// TIA Portal project "instalacja_cieplna_338a_V15_V16" (V16)

(* hardware
DEVICE "GSD device_1"  GSD.Device.PN
   slot 0: "Rack"  Rail  V1.0
   slot 0: "AL1102_2"  AL1102
   slot 1: "8 Ports_1"  AL1102
DEVICE "GSD device_2"  GSD.Device.PN
   slot 0: "Rack"  Rail  V1.0
   slot 0: "AL1102_3"  AL1102
   slot 1: "8 Ports_1"  AL1102
DEVICE "GSD device_3"  GSD.Device.PN
   slot 0: "Rack"  Rail  V1.0
   slot 0: "AL1102_4"  AL1102
   slot 1: "8 Ports_1"  AL1102
   slot 6: "IO-Link In  8 Byte + PQI"  IO-Link In  8 Byte + PQI
   slot 8: "IO-Link In  4 Byte + PQI_1"  IO-Link In  4 Byte + PQI
DEVICE "S71500/ET200MP station_2"  S7-1500 station
   slot 0: "Rail_0"  Rack  6ES7 590-1***0-0AA0
   slot 1: "IO device_1"  IM 155-5 PN HF  6ES7 155-5AA00-0AC0  V3.0
   slot 2: "DQ 32x24VDC/0.5A ST_1"  DQ 32x24VDC/0.5A ST  6ES7 522-1BL00-0AB0  V2.0
   slot 3: "AI 8xU/I/RTD/TC ST_1"  AI 8xU/I/RTD/TC ST  6ES7 531-7KF00-0AB0  V2.0
   slot 4: "AQ 4xU/I ST_1"  AQ 4xU/I ST  6ES7 532-5HD00-0AB0  V2.0
DEVICE "S7-1200 station_1"  S7-1200 Station
   slot 0: "Rack_0"  S7-1200 Rack  Rack  V1.0
   slot 1: "PLC_1"  CPU 1212C DC/DC/DC  6ES7 212-1AE40-0XB0  V4.4
*)

// ===== PLC "PLC_1"  CPU 1212C DC/DC/DC =====

VAR_GLOBAL   // PLC tag table "Default tag table"
   "Heater_PWR_Out" AT %Q0.3 : Bool;
   "Heater_Tout_In" AT %IW127 : Int;   // Temperatura wyjsciowa piec
   "HeatEx_1_Tin_1_In" AT %IW35 : Int;   // Tin wym gora ciepła
   "HeatEx_1_Tout_1_In" AT %IW83 : Int;   // Tout wym gora ciepła
   "Heater_Flow_In" AT %IW112 : Int;   // Przepływ na wejsciu do ogrzewacza
   "HeatEx_1_Flow_In" AT %IW40 : Int;   // przepływ F2
   "Heater_Tin_In" AT %IW103 : Int;   // Temperatura wejściowa piec
   "Heater_Valve_Out" AT %QW8 : Int;   // Wyjście na zawór piec
   "HeatEx_1_Valve_Out" AT %QW4 : Int;   // Wyjscie na zawor wymiennika ciepla góra
   "HeatEx_1_Tin_2_In" AT %IW78 : Int;   // Tin wym gora zimna
   "HeatEx_1_Tout_2_In" AT %IW30 : Int;   // Tout wym gora zimna
   "HeatEx_2_Tin_2_In" AT %IW73 : Int;   // Tin wym dol zimna
   "HeatEx_2_Tin_1_In" AT %IW68 : Int;   // Tin wym dol ciepła
   "HeatEx_2_Tout_2_In" AT %IW122 : Int;   // Tout wym dol zimna
   "HeatEx_2_ValveOut" AT %QW6 : Int;   // wyjście na zawór wymiennika ciepła dół
   "HeatEx_2_Flow_In" AT %IW49 : Int;   // przepływ F3
   "Preassure_In" AT %IW132 : Int;   // Cisnienie wejsciowe na piec
   "off" AT %M0.0 : Bool;
   "start" AT %M0.1 : Bool;
   "reset" AT %M0.2 : Bool;
   "dist" AT %MD2 : Real;
   "dist_SP" AT %MD6 : Real;
   "test" AT %MD10 : Real;
   "step_dist" AT %MD14 : Real;
   "HeatEx_SP" AT %MD18 : Real;
   "HeatEx_2_Tout1_In" AT %IW98 : Int;   // Tout wym dol ciepła
   "Always_OFF" AT %M0.3 : Bool;
   "Preassure_HeatEx_In" AT %IW11 : Int;
   "Preassure_HeatEx_Out" AT %IW17 : Int;
   "Tag_1" AT %QW1 : Int;
   "Tag_2" AT %QW0 : Int;
END_VAR

VAR_GLOBAL CONSTANT   // PLC tag table "Default tag table"
   "None(1)" : Pip := 65535;
   "Automatic update(1)" : Pip := 0;
   "PIP 1(1)" : Pip := 1;
   "PIP 2(1)" : Pip := 2;
   "PIP 3(1)" : Pip := 3;
   "PIP 4(1)" : Pip := 4;
   "PIP 5" : Pip := 5;
   "PIP 6" : Pip := 6;
   "PIP 7" : Pip := 7;
   "PIP 8" : Pip := 8;
   "PIP 9" : Pip := 9;
   "PIP 10" : Pip := 10;
   "PIP 11" : Pip := 11;
   "PIP 12" : Pip := 12;
   "PIP 13" : Pip := 13;
   "PIP 14" : Pip := 14;
   "PIP 15" : Pip := 15;
   "PIP 16" : Pip := 16;
   "PIP 17" : Pip := 17;
   "PIP 18" : Pip := 18;
   "PIP 19" : Pip := 19;
   "PIP 20" : Pip := 20;
   "PIP 21" : Pip := 21;
   "PIP 22" : Pip := 22;
   "PIP 23" : Pip := 23;
   "PIP 24" : Pip := 24;
   "PIP 25" : Pip := 25;
   "PIP 26" : Pip := 26;
   "PIP 27" : Pip := 27;
   "PIP 28" : Pip := 28;
   "PIP 29" : Pip := 29;
   "PIP 30" : Pip := 30;
   "PIP 31" : Pip := 31;
   "PIP OB Servo(1)" : Pip := 32768;
   "Local~Common(1)" : Hw_SubModule := 50;
   "Local(1)" : Hw_SubModule := 49;
   "OB_Main(1)" : OB_PCYCLE := 1;
   "Local~Display" : Hw_SubModule := 54;
   "Local~MC(1)" : Hw_SubModule := 51;
   "Local~Exec(1)" : Hw_SubModule := 52;
   "Local~PROFINET_interface_1(1)" : Hw_Interface := 64;
   "Local~PROFINET_interface_1~Port_1(1)" : Hw_Interface := 65;
   "Local~PROFINET_interface_1~Port_2" : Hw_Interface := 66;
   "Local~PROFINET_IO-System" : Hw_IoSystem := 257;
   "AL1102_4~Proxy" : Hw_SubModule := 310;
   "AL1102_4~IODevice" : Hw_Device := 308;
   "AL1102_4~X1" : Hw_Interface := 311;
   "AL1102_4~X1~Port_1" : Hw_Interface := 312;
   "AL1102_4~X1~Port_2" : Hw_Interface := 283;
   "AL1102_4~Head" : Hw_SubModule := 284;
   "AL1102_4~8_Ports_1~IO-Link_Master" : Hw_SubModule := 286;
   "AL1102_4~8_Ports_1" : Hw_SubModule := 303;
   "AL1102_4~8_Ports_1~IO-Link_In__4_Byte_+_PQI" : Hw_SubModule := 304;
   "AL1102_4~8_Ports_1~IO-Link_In__8_Byte_+_PQI" : Hw_SubModule := 305;
   "AL1102_4~8_Ports_1~IO-Link_In__4_Byte_+_PQI_2" : Hw_SubModule := 307;
   "AL1102_3~Proxy" : Hw_SubModule := 280;
   "AL1102_3~IODevice" : Hw_Device := 278;
   "AL1102_3~X1" : Hw_Interface := 281;
   "AL1102_3~X1~Port_1" : Hw_Interface := 282;
   "AL1102_3~X1~Port_2" : Hw_Interface := 276;
   "AL1102_3~Head" : Hw_SubModule := 277;
   "AL1102_3~8_Ports_1~IO-Link_Master" : Hw_SubModule := 287;
   "AL1102_3~8_Ports_1" : Hw_SubModule := 292;
   "AL1102_3~8_Ports_1~IO-Link_In__8_Byte_+_PQI" : Hw_SubModule := 293;
   "AL1102_3~8_Ports_1~IO-Link_In__8_Byte_+_PQI_1" : Hw_SubModule := 294;
   "AL1102_3~8_Ports_1~IO-Link_In__4_Byte_+_PQI" : Hw_SubModule := 295;
   "AL1102_3~8_Ports_1~IO-Link_In__4_Byte_+_PQI_1" : Hw_SubModule := 296;
   "AL1102_3~8_Ports_1~IO-Link_In__4_Byte_+_PQI_2" : Hw_SubModule := 297;
   "AL1102_3~8_Ports_1~IO-Link_In__4_Byte_+_PQI_3" : Hw_SubModule := 298;
   "AL1102_2~Proxy" : Hw_SubModule := 273;
   "AL1102_2~IODevice" : Hw_Device := 271;
   "AL1102_2~PROFINET_interface_1" : Hw_Interface := 274;
   "AL1102_2~PROFINET_interface_1~Port_1" : Hw_Interface := 268;
   "AL1102_2~PROFINET_interface_1~Port_2" : Hw_Interface := 269;
   "AL1102_2~Head" : Hw_SubModule := 270;
   "AL1102_2~8_Ports_1~IO-Link_Master" : Hw_SubModule := 275;
   "AL1102_2~8_Ports_1~IO-Link_In__4_Byte_+_PQI" : Hw_SubModule := 288;
   "AL1102_2~8_Ports_1" : Hw_SubModule := 285;
   "AL1102_2~8_Ports_1~IO-Link_In__4_Byte_+_PQI_1" : Hw_SubModule := 289;
   "AL1102_2~8_Ports_1~IO-Link_In__4_Byte_+_PQI_2" : Hw_SubModule := 290;
   "AL1102_2~8_Ports_1~IO-Link_In__4_Byte_+_PQI_3" : Hw_SubModule := 291;
   "AL1102_2~8_Ports_1~IO-Link_In__4_Byte_+_PQI_4" : Hw_SubModule := 299;
   "AL1102_2~8_Ports_1~IO-Link_In__4_Byte_+_PQI_5" : Hw_SubModule := 300;
   "AL1102_2~8_Ports_1~IO-Link_In__4_Byte_+_PQI_7" : Hw_SubModule := 302;
   "IO_device_1~Proxy" : Hw_SubModule := 315;
   "IO_device_1~IODevice" : Hw_Device := 313;
   "IO_device_1~PROFINET_interface" : Hw_Interface := 316;
   "IO_device_1~PROFINET_interface~Port_1" : Hw_Interface := 317;
   "IO_device_1~PROFINET_interface~Port_2" : Hw_Interface := 318;
   "IO_device_1~Head" : Hw_SubModule := 319;
   "IO_device_1~DQ_32x24VDC_0_5A_ST_1" : Hw_SubModule := 320;
   "IO_device_1~AI_8xU_I_RTD_TC_ST_1" : Hw_SubModule := 321;
   "IO_device_1~AQ_4xU_I_ST_1" : Hw_SubModule := 322;
   "OB_Startup(1)" : OB_STARTUP := 100;
   "OB_Flow controllers(1)" : OB_Cyclic := 30;
END_VAR

DATA_BLOCK "Signals_DB"   // DB3
{ S7_Optimized_Access := 'TRUE' }
VERSION : 0.1
   VAR
      Heater_Tout_PIDOut : Real;
      Heater_Tout_SP : Real;
      PWM_period : Int;
      PIorPID : Bool;   // 0 - PI, 1 - PID
      Heater_PWR : Real;
      Heater_Alarm : Bool;
      Heater_ResetAlarm : Bool;
      Heater_Tin : Real;
   END_VAR
   VAR RETAIN
      Heater_Tout : Real;
   END_VAR
   VAR
      HeatEx_1_Tin_1 : Real;
      HeatEx_1_Tin_2 : Real;
      HeatEx_1_Tout_1 : Real;
      HeatEx_1_Tout_2 : Real;
      HeatEx_2_Tin_1 : Real;
      HeatEx_2_Tin_2 : Real;
      HeatEx_2_Tout_1 : Real;
      HeatEx_2_Tout_2 : Real;
      Heater_Flow : Real;
      HeatEx_1_Flow : Real;
      HeatEx_2_Flow : Real;
      Heater_Flow_SP : Real;
      Heater_Valve : Real;
      Preassure : Real;
      Preassure_HeatEx_In : Real;
      Preassure_HeatEx_Out : Real;
      HeatEx_1_Flow_SP : Real;
      HeatEx_1_Valve : Real;
      HeatEx_2_FlowSP : Real;
      HeatEx_2_Valve : Real;
      AutoOrManual : Bool;   // Manual = true, Auto = false
      Tout_setpoint : Real;
      PIDMode : Int := 3;
   END_VAR
BEGIN
END_DATA_BLOCK

DATA_BLOCK "PWM_DB"   // DB6
{ S7_Optimized_Access := 'TRUE' }
VERSION : 0.1
// stored: InstanceOfName PWM
"PWM"
BEGIN
END_DATA_BLOCK

DATA_BLOCK "Signals_to_S7protocol"   // DB8
{ S7_Optimized_Access := 'FALSE' }
VERSION : 0.1
   VAR
      OUT : Struct   // PLC out going to Raspbery
         Heater_Tout_setpoint : Real;   // Setpoint output temperature [°C]
         Heater_Flow_actual : Real;   // Actual flow [l/min]
         Heater_Flow_setpoint : Real;   // Flow setpoint[l/min]
         Auto_Or_Manual : Bool;   // Auto - true MAnual - false
         Heater_Tout_actual : Real;   // Actual output temperature [°C]
         Heater_Power_setpoint : Real;   // Percentage heater power rate 0-100
         Counter_OUT : Int;   // Output counter to Raspberry PI
      END_STRUCT;
      IN : Struct   // PLC in from Raspberry
         Flow_setpoint : Real;   // Flow setpoint [l/min]
         Counter_IN : Int;   // Input ciunter from Raspberry PI
      END_STRUCT;
      IN_OUT : Struct
         LiveBit : Bool;   // Communication LiveBit setting in each cycle of OB32
      END_STRUCT;
      INTERNAL : Struct
         Communication_Error : Bool;   // Communication error alarm
         Count_Up_Each_Cycle : Bool;
      END_STRUCT;
   END_VAR
BEGIN
END_DATA_BLOCK

// folder: System blocks/Program resources

DATA_BLOCK "IEC_Timer_0_DB"   // DB1
{ S7_Optimized_Access := 'TRUE' }
AUTHOR : Simatic
FAMILY : IEC
NAME : IEC_TMR
VERSION : 1.0
// stored: InstanceOfName IEC_TIMER
"IEC_TIMER"
BEGIN
END_DATA_BLOCK

DATA_BLOCK "IEC_Timer_0_DB_1"   // DB2
{ S7_Optimized_Access := 'TRUE' }
AUTHOR : Simatic
FAMILY : IEC
NAME : IEC_TMR
VERSION : 1.0
// stored: InstanceOfName IEC_TIMER
"IEC_TIMER"
BEGIN
END_DATA_BLOCK

DATA_BLOCK "LiveBit_timer"   // DB9
{ S7_Optimized_Access := 'TRUE' }
AUTHOR : Simatic
FAMILY : IEC
NAME : IEC_TMR
VERSION : 1.0
// stored: InstanceOfName IEC_TIMER
"IEC_TIMER"
BEGIN
END_DATA_BLOCK

DATA_BLOCK "Communication_Couter"   // DB10
{ S7_Optimized_Access := 'TRUE' }
AUTHOR : Simatic
FAMILY : IEC
NAME : CNTR
VERSION : 1.0
// stored: InstanceOfName IEC_COUNTER
"IEC_COUNTER"
BEGIN
END_DATA_BLOCK

// folder: (top level)

FUNCTION_BLOCK "PWM"   // FB2, LAD
{ S7_Optimized_Access := 'TRUE' }
VERSION : 0.1
   VAR_INPUT
      width : Int;
      cycle : Int;
   END_VAR
   VAR_IN_OUT
      output : Bool;
   END_VAR
   VAR_TEMP
      T1 : Int;
      T2 : Int;
      czas1 : Time;
      czas2 : Time;
   END_VAR
BEGIN

REGION Network 1: Obliczanie T1 i T2 na podstawie czasu cyklu i szerokości impulsu
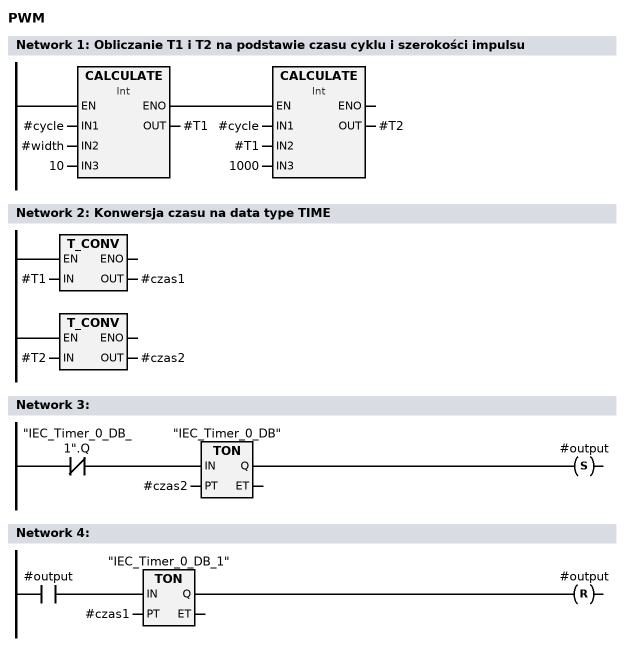
   RUNG wire#powerrail
      { S7_Templates := "SrcType := Int"; S7_GenerateENO := "TRUE"; S7_Expression := "IN1*IN2*IN3" } Calculate(in1 := #cycle, in2 := #width, in3 := 10, out => #T1)
      { S7_Templates := "SrcType := Int"; S7_GenerateENO := "TRUE"; S7_Expression := "IN1*IN3-IN2" } Calculate(in1 := #cycle, in2 := #T1, in3 := 1000, out => #T2)
   END_RUNG
   // the same network as SCL:
   // ENO of a box is taken as its EN; it also drops when the box reports an error
   #T1 := #cycle*#width*10;
   #T2 := #cycle*1000-#T1;
END_REGION

REGION Network 2: Konwersja czasu na data type TIME
   #czas1 := T_CONV(IN := #T1);
   #czas2 := T_CONV(IN := #T2);
END_REGION

REGION Network 3
   "IEC_Timer_0_DB".TON(IN := NOT "IEC_Timer_0_DB_1".Q, PT := #czas2);
   IF "IEC_Timer_0_DB".Q THEN #output := TRUE; END_IF;
END_REGION

REGION Network 4
   "IEC_Timer_0_DB_1".TON(IN := #output, PT := #czas1);
   IF "IEC_Timer_0_DB_1".Q THEN #output := FALSE; END_IF;
END_REGION
END_FUNCTION_BLOCK

ORGANIZATION_BLOCK "Main"   // OB1, LAD, ProgramCycle
TITLE = "Main Program Sweep (Cycle)"
{ S7_Optimized_Access := 'TRUE' }
VERSION : 0.1
   VAR_INPUT
      Initial_Call : Bool;   // Initial call of this OB
      Remanence : Bool;   // =True, if remanent data are available
   END_VAR
   VAR_TEMP
      power_SP_int : Int;
      ret_value : Int;
      scale_press_Heat_Ex_OUT : Real;
      scale_press_PressureIN : Real;
      scale_press_Heat_Ex_IN : Real;
      unscale_Heater_Valve : Real;
      unscale_HeatEX_2_ValveOut : Real;
      unscale_HeatEX_1_ValveOut : Real;
      tmp_PID_Tout_Rate : Real;
   END_VAR
BEGIN

REGION Network 1: Sterowanie mocą pieca
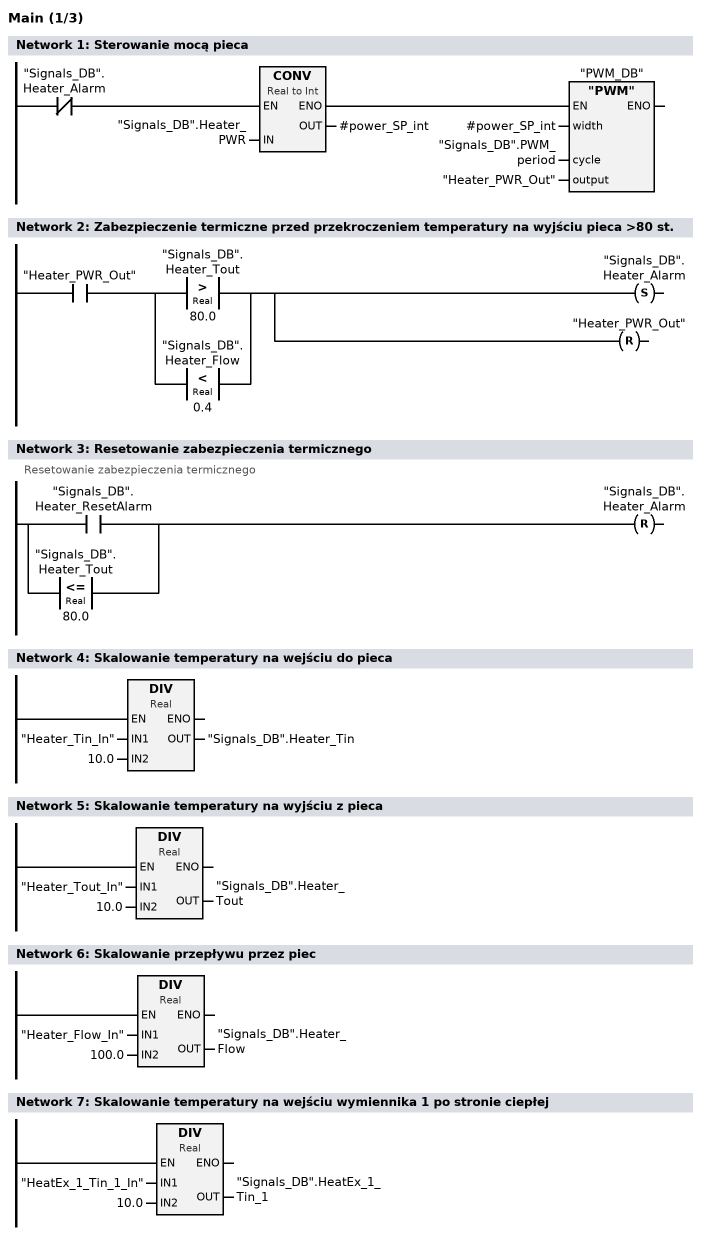
   RUNG wire#powerrail
      I_Contact( "Signals_DB".Heater_Alarm )
      { S7_Templates := "[SrcType := Real, DestType := Int]"; S7_GenerateENO := "TRUE" } Convert(in := "Signals_DB".Heater_PWR, out => #power_SP_int)
      "PWM_DB"(width := #power_SP_int, cycle := "Signals_DB".PWM_period, output := "Heater_PWR_Out")
   END_RUNG
   // the same network as SCL:
   // ENO of a box is taken as its EN; it also drops when the box reports an error
   IF NOT "Signals_DB".Heater_Alarm THEN
       #power_SP_int := REAL_TO_INT("Signals_DB".Heater_PWR);
       "PWM_DB"(width := #power_SP_int, cycle := "Signals_DB".PWM_period, output := "Heater_PWR_Out");   // "PWM"
   END_IF;
END_REGION

REGION Network 2: Zabezpieczenie termiczne przed przekroczeniem temperatury na wyjściu pieca >80 st.
   RUNG wire#powerrail
      Contact( "Heater_PWR_Out" )
      wire#w1
      { S7_Templates := "SrcType := Real" } GT_Contact(in1 := "Signals_DB".Heater_Tout, in2 := 80.0)
      wire#w2
      S_Coil( "Signals_DB".Heater_Alarm )
   END_RUNG
   RUNG wire#w1
      { S7_Templates := "SrcType := Real" } LT_Contact(in1 := "Signals_DB".Heater_Flow, in2 := 0.4)
   END_RUNG wire#w2
   RUNG wire#w2
      R_Coil( "Heater_PWR_Out" )
   END_RUNG
   // the same network as SCL:
   IF "Heater_PWR_Out" AND (("Signals_DB".Heater_Tout > 80.0) OR ("Signals_DB".Heater_Flow < 0.4)) THEN
       "Signals_DB".Heater_Alarm := TRUE;
       "Heater_PWR_Out" := FALSE;
   END_IF;
END_REGION

REGION Network 3: Resetowanie zabezpieczenia termicznego
   // Resetowanie zabezpieczenia termicznego
   RUNG wire#powerrail
      Contact( "Signals_DB".Heater_ResetAlarm )
      wire#w1
      R_Coil( "Signals_DB".Heater_Alarm )
   END_RUNG
   RUNG wire#powerrail
      { S7_Templates := "SrcType := Real" } LE_Contact(in1 := "Signals_DB".Heater_Tout, in2 := 80.0)
   END_RUNG wire#w1
   // the same network as SCL:
   IF "Signals_DB".Heater_ResetAlarm OR ("Signals_DB".Heater_Tout <= 80.0) THEN
       "Signals_DB".Heater_Alarm := FALSE;
   END_IF;
END_REGION

REGION Network 4: Skalowanie temperatury na wejściu do pieca
   RUNG wire#powerrail
      { S7_Templates := "SrcType := Real"; S7_GenerateENO := "TRUE" } Div(in1 := "Heater_Tin_In", in2 := 10.0, out => "Signals_DB".Heater_Tin)
   END_RUNG
   // the same network as SCL:
   "Signals_DB".Heater_Tin := "Heater_Tin_In" / 10.0;
END_REGION

REGION Network 5: Skalowanie temperatury na wyjściu z pieca
   RUNG wire#powerrail
      { S7_Templates := "SrcType := Real"; S7_GenerateENO := "TRUE" } Div(in1 := "Heater_Tout_In", in2 := 10.0, out => "Signals_DB".Heater_Tout)
   END_RUNG
   // the same network as SCL:
   "Signals_DB".Heater_Tout := "Heater_Tout_In" / 10.0;
END_REGION

REGION Network 6: Skalowanie przepływu przez piec
   RUNG wire#powerrail
      { S7_Templates := "SrcType := Real"; S7_GenerateENO := "TRUE" } Div(in1 := "Heater_Flow_In", in2 := 100.0, out => "Signals_DB".Heater_Flow)
   END_RUNG
   // the same network as SCL:
   "Signals_DB".Heater_Flow := "Heater_Flow_In" / 100.0;
END_REGION

REGION Network 7: Skalowanie temperatury na wejściu wymiennika 1 po stronie ciepłej
   RUNG wire#powerrail
      { S7_Templates := "SrcType := Real"; S7_GenerateENO := "TRUE" } Div(in1 := "HeatEx_1_Tin_1_In", in2 := 10.0, out => "Signals_DB".HeatEx_1_Tin_1)
   END_RUNG
   // the same network as SCL:
   "Signals_DB".HeatEx_1_Tin_1 := "HeatEx_1_Tin_1_In" / 10.0;
END_REGION

REGION Network 8: Skalowanie temperatury na wyjściu z wymiennika 1 po stronie ciepłej
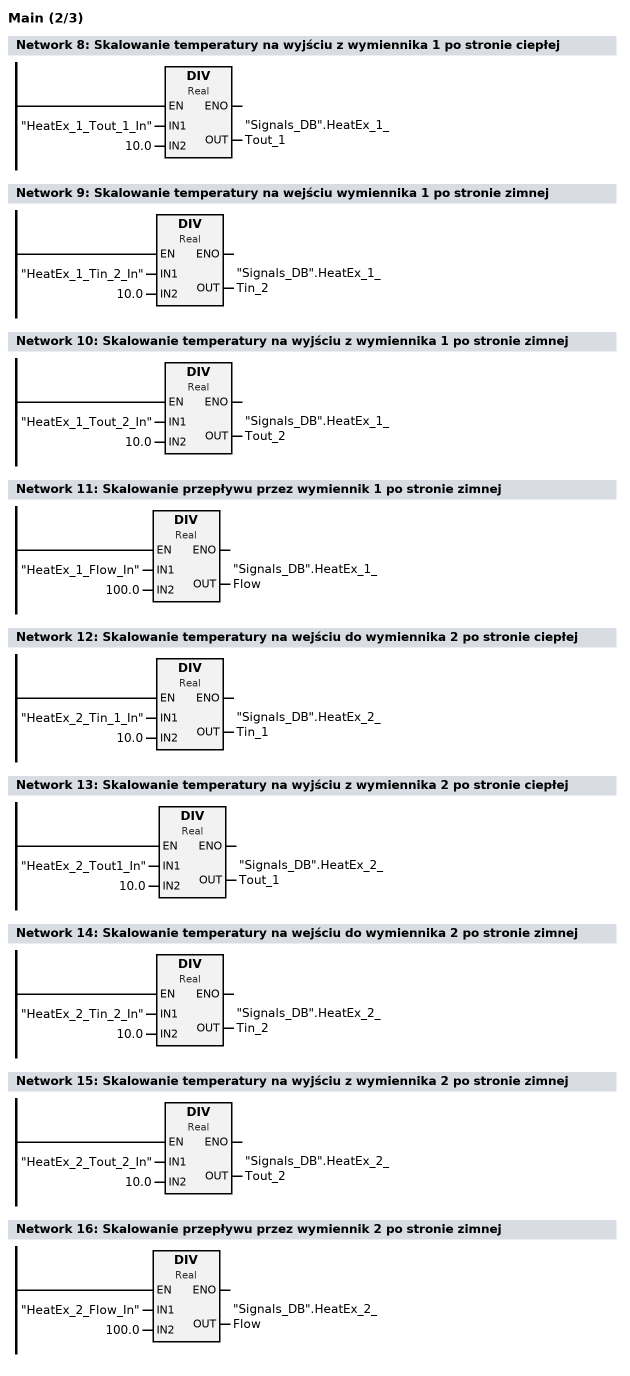
   RUNG wire#powerrail
      { S7_Templates := "SrcType := Real"; S7_GenerateENO := "TRUE" } Div(in1 := "HeatEx_1_Tout_1_In", in2 := 10.0, out => "Signals_DB".HeatEx_1_Tout_1)
   END_RUNG
   // the same network as SCL:
   "Signals_DB".HeatEx_1_Tout_1 := "HeatEx_1_Tout_1_In" / 10.0;
END_REGION

REGION Network 9: Skalowanie temperatury na wejściu wymiennika 1 po stronie zimnej
   RUNG wire#powerrail
      { S7_Templates := "SrcType := Real"; S7_GenerateENO := "TRUE" } Div(in1 := "HeatEx_1_Tin_2_In", in2 := 10.0, out => "Signals_DB".HeatEx_1_Tin_2)
   END_RUNG
   // the same network as SCL:
   "Signals_DB".HeatEx_1_Tin_2 := "HeatEx_1_Tin_2_In" / 10.0;
END_REGION

REGION Network 10: Skalowanie temperatury na wyjściu z wymiennika 1 po stronie zimnej
   RUNG wire#powerrail
      { S7_Templates := "SrcType := Real"; S7_GenerateENO := "TRUE" } Div(in1 := "HeatEx_1_Tout_2_In", in2 := 10.0, out => "Signals_DB".HeatEx_1_Tout_2)
   END_RUNG
   // the same network as SCL:
   "Signals_DB".HeatEx_1_Tout_2 := "HeatEx_1_Tout_2_In" / 10.0;
END_REGION

REGION Network 11: Skalowanie przepływu przez wymiennik 1 po stronie zimnej
   RUNG wire#powerrail
      { S7_Templates := "SrcType := Real"; S7_GenerateENO := "TRUE" } Div(in1 := "HeatEx_1_Flow_In", in2 := 100.0, out => "Signals_DB".HeatEx_1_Flow)
   END_RUNG
   // the same network as SCL:
   "Signals_DB".HeatEx_1_Flow := "HeatEx_1_Flow_In" / 100.0;
END_REGION

REGION Network 12: Skalowanie temperatury na wejściu do wymiennika 2 po stronie ciepłej
   RUNG wire#powerrail
      { S7_Templates := "SrcType := Real"; S7_GenerateENO := "TRUE" } Div(in1 := "HeatEx_2_Tin_1_In", in2 := 10.0, out => "Signals_DB".HeatEx_2_Tin_1)
   END_RUNG
   // the same network as SCL:
   "Signals_DB".HeatEx_2_Tin_1 := "HeatEx_2_Tin_1_In" / 10.0;
END_REGION

REGION Network 13: Skalowanie temperatury na wyjściu z wymiennika 2 po stronie ciepłej
   RUNG wire#powerrail
      { S7_Templates := "SrcType := Real"; S7_GenerateENO := "TRUE" } Div(in1 := "HeatEx_2_Tout1_In", in2 := 10.0, out => "Signals_DB".HeatEx_2_Tout_1)
   END_RUNG
   // the same network as SCL:
   "Signals_DB".HeatEx_2_Tout_1 := "HeatEx_2_Tout1_In" / 10.0;
END_REGION

REGION Network 14: Skalowanie temperatury na wejściu do wymiennika 2 po stronie zimnej
   RUNG wire#powerrail
      { S7_Templates := "SrcType := Real"; S7_GenerateENO := "TRUE" } Div(in1 := "HeatEx_2_Tin_2_In", in2 := 10.0, out => "Signals_DB".HeatEx_2_Tin_2)
   END_RUNG
   // the same network as SCL:
   "Signals_DB".HeatEx_2_Tin_2 := "HeatEx_2_Tin_2_In" / 10.0;
END_REGION

REGION Network 15: Skalowanie temperatury na wyjściu z wymiennika 2 po stronie zimnej
   RUNG wire#powerrail
      { S7_Templates := "SrcType := Real"; S7_GenerateENO := "TRUE" } Div(in1 := "HeatEx_2_Tout_2_In", in2 := 10.0, out => "Signals_DB".HeatEx_2_Tout_2)
   END_RUNG
   // the same network as SCL:
   "Signals_DB".HeatEx_2_Tout_2 := "HeatEx_2_Tout_2_In" / 10.0;
END_REGION

REGION Network 16: Skalowanie przepływu przez wymiennik 2 po stronie zimnej
   RUNG wire#powerrail
      { S7_Templates := "SrcType := Real"; S7_GenerateENO := "TRUE" } Div(in1 := "HeatEx_2_Flow_In", in2 := 100.0, out => "Signals_DB".HeatEx_2_Flow)
   END_RUNG
   // the same network as SCL:
   "Signals_DB".HeatEx_2_Flow := "HeatEx_2_Flow_In" / 100.0;
END_REGION

REGION Network 17: Unskalowanie otwarcia zaworu wyjściowego z pieca
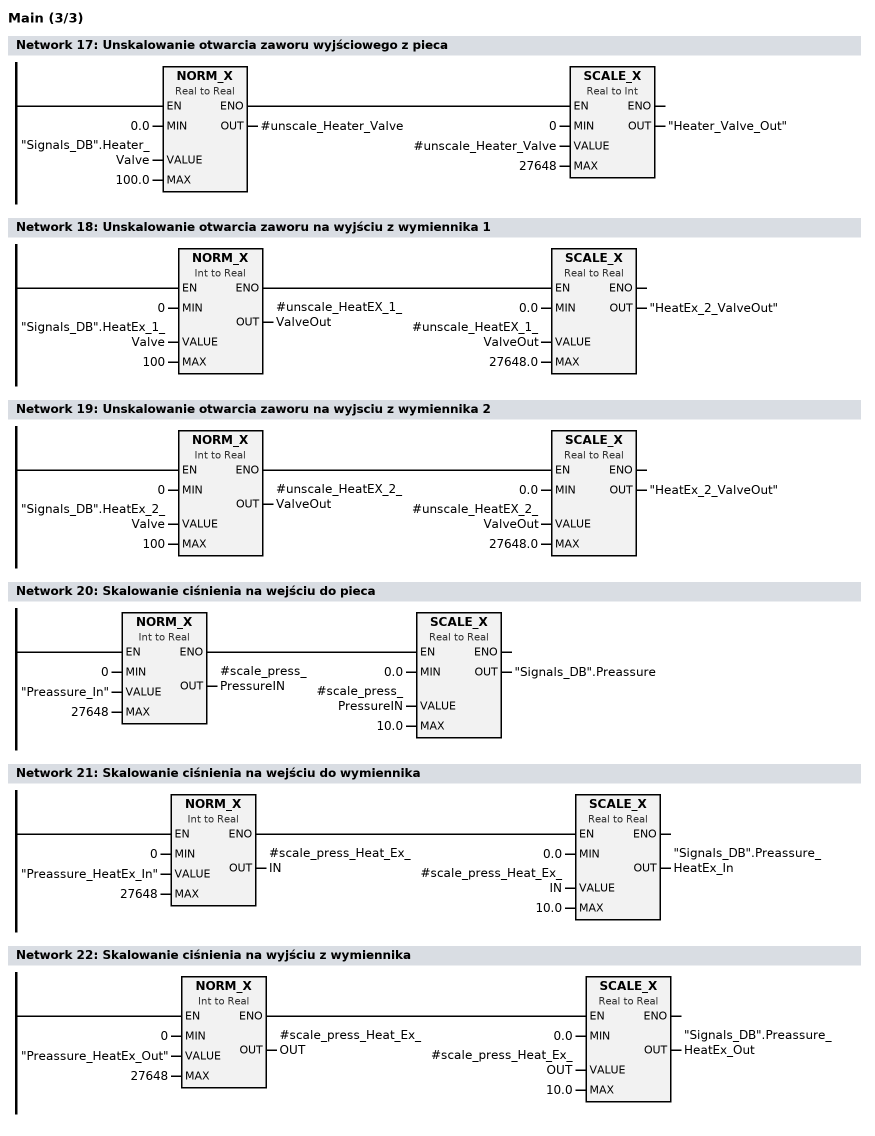
   RUNG wire#powerrail
      { S7_Templates := "[SrcType := Real, DestType := Real]" } Normalize(min := 0.0, value := "Signals_DB".Heater_Valve, max := 100.0, out => #unscale_Heater_Valve)
      { S7_Templates := "[SrcType := Real, DestType := Int]" } Scale(min := 0, value := #unscale_Heater_Valve, max := 27648, out => "Heater_Valve_Out")
   END_RUNG
   // the same network as SCL:
   #unscale_Heater_Valve := NORM_X(MIN := 0.0, VALUE := "Signals_DB".Heater_Valve, MAX := 100.0);
   "Heater_Valve_Out" := SCALE_X(MIN := 0, VALUE := #unscale_Heater_Valve, MAX := 27648);
END_REGION

REGION Network 18: Unskalowanie otwarcia zaworu na wyjściu z wymiennika 1
   RUNG wire#powerrail
      { S7_Templates := "[SrcType := Int, DestType := Real]" } Normalize(min := 0, value := "Signals_DB".HeatEx_1_Valve, max := 100, out => #unscale_HeatEX_1_ValveOut)
      { S7_Templates := "[SrcType := Real, DestType := Real]" } Scale(min := 0.0, value := #unscale_HeatEX_1_ValveOut, max := 27648.0, out => "HeatEx_2_ValveOut")
   END_RUNG
   // the same network as SCL:
   #unscale_HeatEX_1_ValveOut := NORM_X(MIN := 0, VALUE := "Signals_DB".HeatEx_1_Valve, MAX := 100);
   "HeatEx_2_ValveOut" := SCALE_X(MIN := 0.0, VALUE := #unscale_HeatEX_1_ValveOut, MAX := 27648.0);
END_REGION

REGION Network 19: Unskalowanie otwarcia zaworu na wyjsciu z wymiennika 2
   RUNG wire#powerrail
      { S7_Templates := "[SrcType := Int, DestType := Real]" } Normalize(min := 0, value := "Signals_DB".HeatEx_2_Valve, max := 100, out => #unscale_HeatEX_2_ValveOut)
      { S7_Templates := "[SrcType := Real, DestType := Real]" } Scale(min := 0.0, value := #unscale_HeatEX_2_ValveOut, max := 27648.0, out => "HeatEx_2_ValveOut")
   END_RUNG
   // the same network as SCL:
   #unscale_HeatEX_2_ValveOut := NORM_X(MIN := 0, VALUE := "Signals_DB".HeatEx_2_Valve, MAX := 100);
   "HeatEx_2_ValveOut" := SCALE_X(MIN := 0.0, VALUE := #unscale_HeatEX_2_ValveOut, MAX := 27648.0);
END_REGION

REGION Network 20: Skalowanie ciśnienia na wejściu do pieca
   RUNG wire#powerrail
      { S7_Templates := "[SrcType := Int, DestType := Real]" } Normalize(min := 0, value := "Preassure_In", max := 27648, out => #scale_press_PressureIN)
      { S7_Templates := "[SrcType := Real, DestType := Real]" } Scale(min := 0.0, value := #scale_press_PressureIN, max := 10.0, out => "Signals_DB".Preassure)
   END_RUNG
   // the same network as SCL:
   #scale_press_PressureIN := NORM_X(MIN := 0, VALUE := "Preassure_In", MAX := 27648);
   "Signals_DB".Preassure := SCALE_X(MIN := 0.0, VALUE := #scale_press_PressureIN, MAX := 10.0);
END_REGION

REGION Network 21: Skalowanie ciśnienia na wejściu do wymiennika
   RUNG wire#powerrail
      { S7_Templates := "[SrcType := Int, DestType := Real]" } Normalize(min := 0, value := "Preassure_HeatEx_In", max := 27648, out => #scale_press_Heat_Ex_IN)
      { S7_Templates := "[SrcType := Real, DestType := Real]" } Scale(min := 0.0, value := #scale_press_Heat_Ex_IN, max := 10.0, out => "Signals_DB".Preassure_HeatEx_In)
   END_RUNG
   // the same network as SCL:
   #scale_press_Heat_Ex_IN := NORM_X(MIN := 0, VALUE := "Preassure_HeatEx_In", MAX := 27648);
   "Signals_DB".Preassure_HeatEx_In := SCALE_X(MIN := 0.0, VALUE := #scale_press_Heat_Ex_IN, MAX := 10.0);
END_REGION

REGION Network 22: Skalowanie ciśnienia na wyjściu z wymiennika
   RUNG wire#powerrail
      { S7_Templates := "[SrcType := Int, DestType := Real]" } Normalize(min := 0, value := "Preassure_HeatEx_Out", max := 27648, out => #scale_press_Heat_Ex_OUT)
      { S7_Templates := "[SrcType := Real, DestType := Real]" } Scale(min := 0.0, value := #scale_press_Heat_Ex_OUT, max := 10.0, out => "Signals_DB".Preassure_HeatEx_Out)
   END_RUNG
   // the same network as SCL:
   #scale_press_Heat_Ex_OUT := NORM_X(MIN := 0, VALUE := "Preassure_HeatEx_Out", MAX := 27648);
   "Signals_DB".Preassure_HeatEx_Out := SCALE_X(MIN := 0.0, VALUE := #scale_press_Heat_Ex_OUT, MAX := 10.0);
END_REGION
END_ORGANIZATION_BLOCK

ORGANIZATION_BLOCK "Flow controllers"   // OB30, LAD, CyclicInterrupt
{ S7_Optimized_Access := 'TRUE' }
VERSION : 0.1
   VAR_INPUT
      Initial_Call : Bool;   // Initial call of this OB
      Event_Count : Int;   // Events discarded
   END_VAR
   VAR_TEMP
      PIorPID : Bool;
   END_VAR
BEGIN

REGION Network 1: PID do sterowania nagrzewaniem cieczy
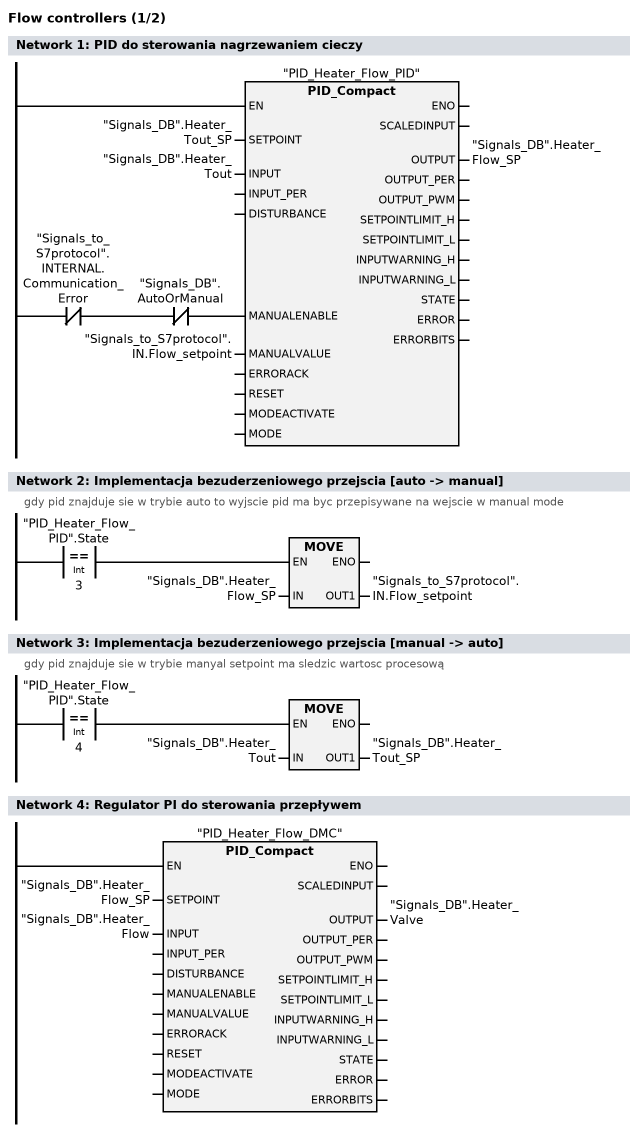
   "PID_Heater_Flow_PID"(Setpoint := "Signals_DB".Heater_Tout_SP,   // PID_Compact
                         Input := "Signals_DB".Heater_Tout,
                         ManualEnable := NOT "Signals_to_S7protocol".INTERNAL.Communication_Error AND NOT "Signals_DB".AutoOrManual,
                         ManualValue := "Signals_to_S7protocol".IN.Flow_setpoint,
                         Output => "Signals_DB".Heater_Flow_SP);
END_REGION

REGION Network 2: Implementacja bezuderzeniowego przejscia [auto -> manual]
   // gdy pid znajduje sie w trybie auto to wyjscie pid ma byc przepisywane na wejscie w manual mode
   RUNG wire#powerrail
      { S7_Templates := "SrcType := Int" } EQ_Contact(in1 := "PID_Heater_Flow_PID".State, in2 := 3)
      Move(in := "Signals_DB".Heater_Flow_SP, out1 => "Signals_to_S7protocol".IN.Flow_setpoint)
   END_RUNG
   // the same network as SCL:
   IF "PID_Heater_Flow_PID".State = 3 THEN
       "Signals_to_S7protocol".IN.Flow_setpoint := "Signals_DB".Heater_Flow_SP;
   END_IF;
END_REGION

REGION Network 3: Implementacja bezuderzeniowego przejscia [manual -> auto]
   // gdy pid znajduje sie w trybie manyal setpoint ma sledzic wartosc procesową
   RUNG wire#powerrail
      { S7_Templates := "SrcType := Int" } EQ_Contact(in1 := "PID_Heater_Flow_PID".State, in2 := 4)
      Move(in := "Signals_DB".Heater_Tout, out1 => "Signals_DB".Heater_Tout_SP)
   END_RUNG
   // the same network as SCL:
   IF "PID_Heater_Flow_PID".State = 4 THEN "Signals_DB".Heater_Tout_SP := "Signals_DB".Heater_Tout; END_IF;
END_REGION

REGION Network 4: Regulator PI do sterowania przepływem
   "PID_Heater_Flow_DMC"(Setpoint := "Signals_DB".Heater_Flow_SP,   // PID_Compact
                         Input := "Signals_DB".Heater_Flow,
                         Output => "Signals_DB".Heater_Valve);
END_REGION

REGION Network 5
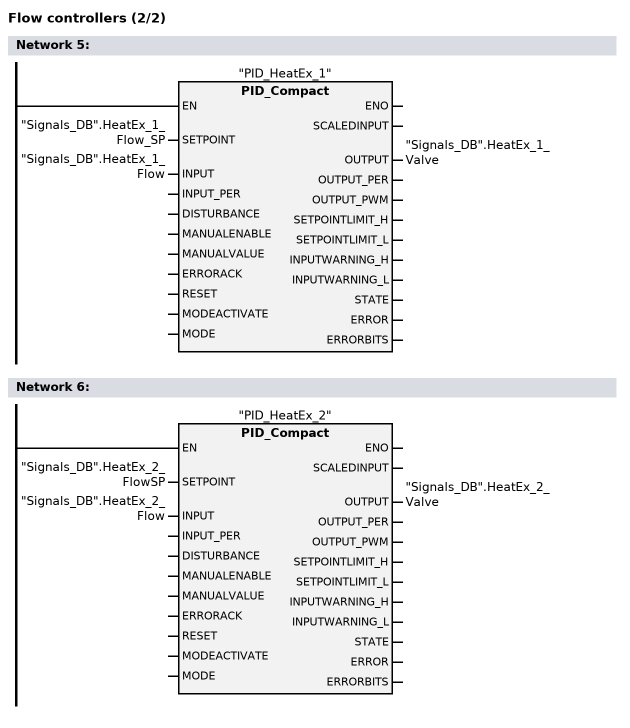
   "PID_HeatEx_1"(Setpoint := "Signals_DB".HeatEx_1_Flow_SP,   // PID_Compact
                  Input := "Signals_DB".HeatEx_1_Flow,
                  Output => "Signals_DB".HeatEx_1_Valve);
END_REGION

REGION Network 6
   "PID_HeatEx_2"(Setpoint := "Signals_DB".HeatEx_2_FlowSP,   // PID_Compact
                  Input := "Signals_DB".HeatEx_2_Flow,
                  Output => "Signals_DB".HeatEx_2_Valve);
END_REGION
END_ORGANIZATION_BLOCK

ORGANIZATION_BLOCK "Scaled rewrite"   // OB32, LAD, CyclicInterrupt
{ S7_Optimized_Access := 'TRUE' }
VERSION : 0.1
   VAR_INPUT
      Initial_Call : Bool;   // Initial call of this OB
      Event_Count : Int;   // Events discarded
   END_VAR
   VAR_TEMP
      time_LiveBit_NOK : Time;
      bool_LiveBit_NOK : Bool;
      bool_Reset_Communication_Counter : Bool;
      "int _Counter_Differance" : Int;
      bool_Count_Up_Each_Cycle_possitive : Bool;
      bool_Count_Up_Each_Cycle_negative : Bool;
      int_Odd_Or_Even : Int;
   END_VAR
BEGIN

REGION Network 1: Flow setpoint to PI
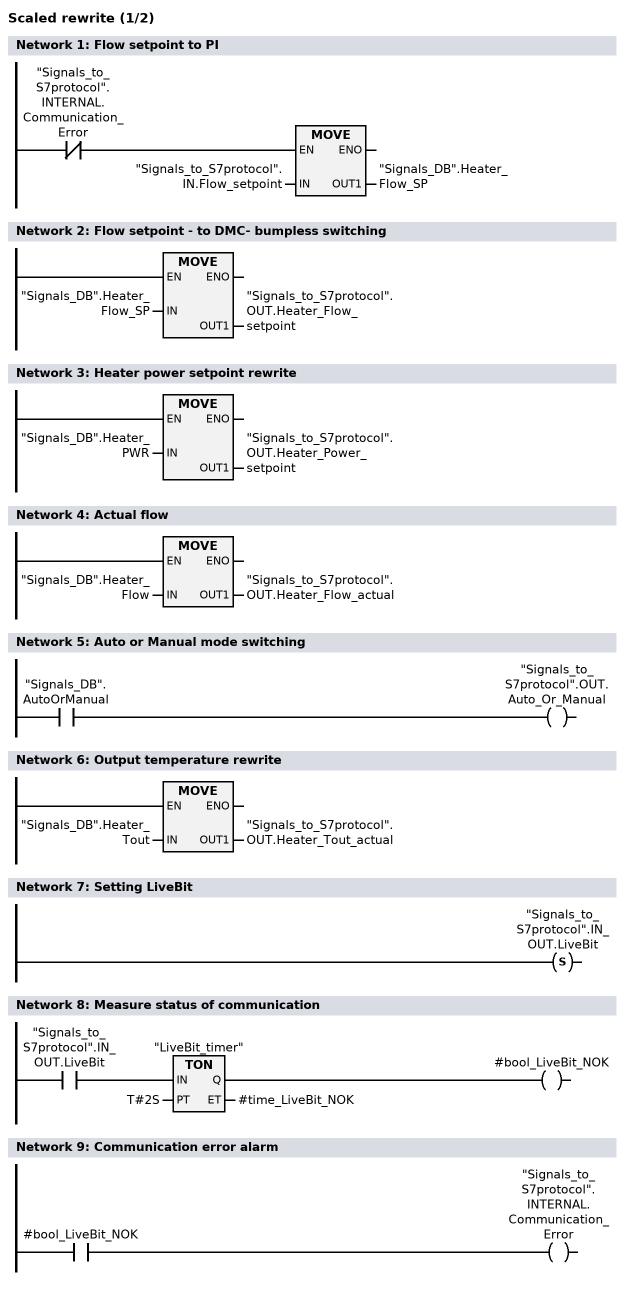
   RUNG wire#powerrail
      I_Contact( "Signals_to_S7protocol".INTERNAL.Communication_Error )
      Move(in := "Signals_to_S7protocol".IN.Flow_setpoint, out1 => "Signals_DB".Heater_Flow_SP)
   END_RUNG
   // the same network as SCL:
   IF NOT "Signals_to_S7protocol".INTERNAL.Communication_Error THEN
       "Signals_DB".Heater_Flow_SP := "Signals_to_S7protocol".IN.Flow_setpoint;
   END_IF;
END_REGION

REGION Network 2: Flow setpoint - to DMC- bumpless switching
   RUNG wire#powerrail
      Move(in := "Signals_DB".Heater_Flow_SP, out1 => "Signals_to_S7protocol".OUT.Heater_Flow_setpoint)
   END_RUNG
   // the same network as SCL:
   "Signals_to_S7protocol".OUT.Heater_Flow_setpoint := "Signals_DB".Heater_Flow_SP;
END_REGION

REGION Network 3: Heater power setpoint rewrite
   RUNG wire#powerrail
      Move(in := "Signals_DB".Heater_PWR, out1 => "Signals_to_S7protocol".OUT.Heater_Power_setpoint)
   END_RUNG
   // the same network as SCL:
   "Signals_to_S7protocol".OUT.Heater_Power_setpoint := "Signals_DB".Heater_PWR;
END_REGION

REGION Network 4: Actual flow
   RUNG wire#powerrail
      Move(in := "Signals_DB".Heater_Flow, out1 => "Signals_to_S7protocol".OUT.Heater_Flow_actual)
   END_RUNG
   // the same network as SCL:
   "Signals_to_S7protocol".OUT.Heater_Flow_actual := "Signals_DB".Heater_Flow;
END_REGION

REGION Network 5: Auto or Manual mode switching
   RUNG wire#powerrail
      Contact( "Signals_DB".AutoOrManual )
      Coil( "Signals_to_S7protocol".OUT.Auto_Or_Manual )
   END_RUNG
   // the same network as SCL:
   "Signals_to_S7protocol".OUT.Auto_Or_Manual := "Signals_DB".AutoOrManual;
END_REGION

REGION Network 6: Output temperature rewrite
   RUNG wire#powerrail
      Move(in := "Signals_DB".Heater_Tout, out1 => "Signals_to_S7protocol".OUT.Heater_Tout_actual)
   END_RUNG
   // the same network as SCL:
   "Signals_to_S7protocol".OUT.Heater_Tout_actual := "Signals_DB".Heater_Tout;
END_REGION

REGION Network 7: Setting LiveBit
   RUNG wire#powerrail
      S_Coil( "Signals_to_S7protocol".IN_OUT.LiveBit )
   END_RUNG
   // the same network as SCL:
   "Signals_to_S7protocol".IN_OUT.LiveBit := TRUE;
END_REGION

REGION Network 8: Measure status of communication
   "LiveBit_timer".TON(IN := "Signals_to_S7protocol".IN_OUT.LiveBit, PT := T#2S, ET => #time_LiveBit_NOK);
   #bool_LiveBit_NOK := "LiveBit_timer".Q;
END_REGION

REGION Network 9: Communication error alarm
   RUNG wire#powerrail
      Contact( #bool_LiveBit_NOK )
      Coil( "Signals_to_S7protocol".INTERNAL.Communication_Error )
   END_RUNG
   // the same network as SCL:
   "Signals_to_S7protocol".INTERNAL.Communication_Error := #bool_LiveBit_NOK;
END_REGION

REGION Network 10: Increment PLC counter
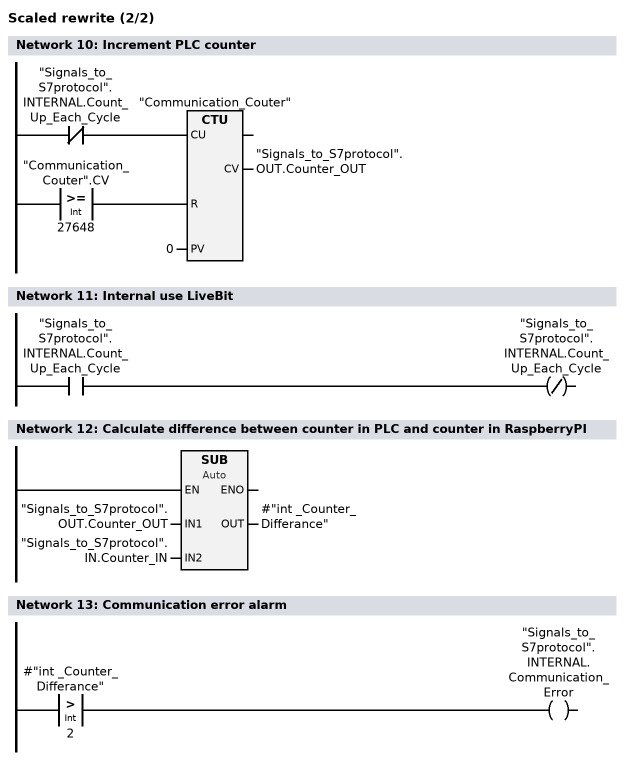
   "Communication_Couter".CTU(CU := NOT "Signals_to_S7protocol".INTERNAL.Count_Up_Each_Cycle,
                           R := "Communication_Couter".CV >= 27648,
                           PV := 0,
                           CV => "Signals_to_S7protocol".OUT.Counter_OUT);
END_REGION

REGION Network 11: Internal use LiveBit
   RUNG wire#powerrail
      Contact( "Signals_to_S7protocol".INTERNAL.Count_Up_Each_Cycle )
      I_Coil( "Signals_to_S7protocol".INTERNAL.Count_Up_Each_Cycle )
   END_RUNG
   // the same network as SCL:
   "Signals_to_S7protocol".INTERNAL.Count_Up_Each_Cycle := NOT "Signals_to_S7protocol".INTERNAL.Count_Up_Each_Cycle;
END_REGION

REGION Network 12: Calculate difference between counter in PLC and counter in RaspberryPI
   RUNG wire#powerrail
      Sub(in1 := "Signals_to_S7protocol".OUT.Counter_OUT, in2 := "Signals_to_S7protocol".IN.Counter_IN, out => #"int _Counter_Differance")
   END_RUNG
   // the same network as SCL:
   #"int _Counter_Differance" := "Signals_to_S7protocol".OUT.Counter_OUT - "Signals_to_S7protocol".IN.Counter_IN;
END_REGION

REGION Network 13: Communication error alarm
   RUNG wire#powerrail
      { S7_Templates := "SrcType := Int" } GT_Contact(in1 := #"int _Counter_Differance", in2 := 2)
      Coil( "Signals_to_S7protocol".INTERNAL.Communication_Error )
   END_RUNG
   // the same network as SCL:
   "Signals_to_S7protocol".INTERNAL.Communication_Error := #"int _Counter_Differance" > 2;
END_REGION
END_ORGANIZATION_BLOCK

ORGANIZATION_BLOCK "Startup"   // OB100, LAD, Startup
TITLE = "Complete Restart"
{ S7_Optimized_Access := 'TRUE' }
VERSION : 0.1
   VAR_INPUT
      LostRetentive : Bool;   // True if retentive data are lost
      LostRTC : Bool;   // True if date and time are lost
   END_VAR
BEGIN

REGION Network 1
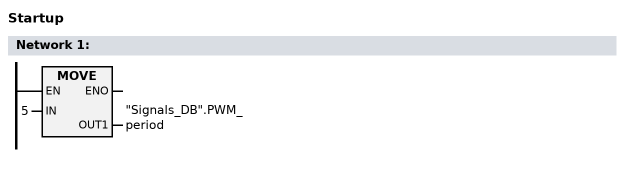
   RUNG wire#powerrail
      { S7_GenerateENO := "TRUE" } Move(in := 5, out1 => "Signals_DB".PWM_period)
   END_RUNG
   // the same network as SCL:
   "Signals_DB".PWM_period := 5;
END_REGION
END_ORGANIZATION_BLOCK